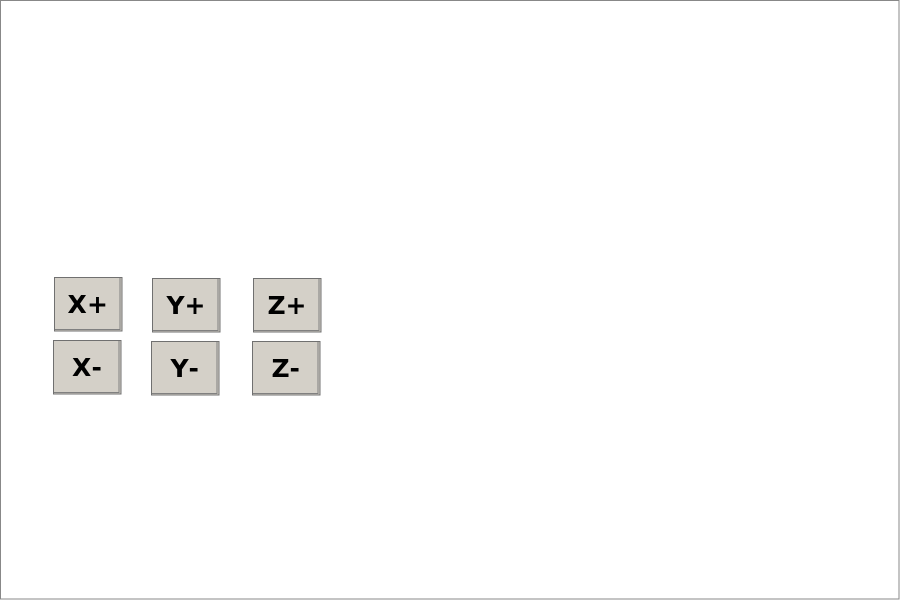
VISUALIZATION Panel  // 900x600
    Button (53,340 68x54), "X-"
        tap GVL.BT_X_AXIS_LEFT
    Button (54,277 68x54), "X+"
        tap GVL.BT_X_AXIS_RIGHT
    Button (152,278 68x54), "Y+"
        tap GVL.BT_Y_AXIS_FRONT
    Button (151,341 68x54), "Y-"
        tap GVL.BT_Y_AXIS_BACK
    Button (253,278 68x54), "Z+"
        tap GVL.Z_AXIS_UP
    Button (252,341 68x54), "Z-"
        tap GVL.Z_AXIS_DOWN
END_VISUALIZATION

(* stored: Version 1.1.0.1, ProductVersion 3.1.4024.13
   Visu Panel: Id {3e8dfa27-72ac-4ed9-8116-e4259ca169ae} *)
